FUNCTION_BLOCK Coche1 EXTENDS Vehiculo
VAR_INPUT
	velocidadMaxima : REAL;
END_VAR
VAR_OUTPUT
END_VAR
VAR
END_VAR


METHOD Mover : REAL
VAR_INPUT
	Velocidad_Deseada : REAL;
END_VAR
Mover := Velocidad_Deseada * velocidadMaxima;
END_METHOD

END_FUNCTION_BLOCK

(* stored: Version 1.1.0.1, ProductVersion 3.1.4024.12
   POU Coche1: Id {cc8ecd1f-0cd7-4903-9c1f-7a7af02f9dfa}, SpecialFunc None
   Method Mover: Id {3881cff0-6e5a-4f89-b566-859812957a0b} *)
